// TIA Portal V19 export
VAR_GLOBAL   // PLC tag table "U2Em5"
END_VAR
VAR_GLOBAL CONSTANT   // user constants
   U2EM5_JOB_EXECUTE : DInt := 100;
   U2EM5_JOB_STOPPING : DInt := 200;
   U2EM5_JOB_HOLODING : DInt := 300;
   U2EM5_JOB_UNHOLODING : DInt := 400;
   U2EM5_JOB_RESTING : DInt := 500;
   U2EM5_JOB_STARTING : DInt := 600;
END_VAR
